PROGRAM GUI_logic
VAR
END_VAR

(*
//Main screen GUI buttons
IF GVL_GUI.main_button_logic THEN
	GVL_GUI.conv_button_logic:= 0;
	GVL_GUI.pcontrol_button_logic:= 0;
	GVL_GUI.qcontrol_button_logic:= 0;
	GVL_GUI.meter_cfg_button_logic:= 0;
ELSIF GVL_GUI.pcontrol_button_logic THEN
	GVL_GUI.main_button_logic:= 0;
	GVL_GUI.conv_button_logic:= 0;
	GVL_GUI.qcontrol_button_logic:= 0;
	GVL_GUI.meter_cfg_button_logic:= 0;
ELSE
	GVL_GUI.main_button_logic:= 0;
	GVL_GUI.conv_button_logic:= 0;
	GVL_GUI.pcontrol_button_logic:= 0;
	GVL_GUI.qcontrol_button_logic:= 0;
	GVL_GUI.meter_cfg_button_logic:= 0;
END_IF
*)

END_PROGRAM

(* stored: Version 1.1.0.1, ProductVersion 3.1.4024.11
   POU GUI_logic: Id {268f483e-8f52-47db-a3dd-9461ababddf0}, SpecialFunc None *)
